// TIA Portal V17 export
// export: Created 2025-07-13T07:45:38.0095536Z, ExportSetting WithDefaults, DisplayName Totally Integrated Automation Portal, DisplayVersion V17, DisplayName TIA Portal Openness, DisplayVersion V17, DisplayName TIA Portal Version Control Interface, DisplayVersion V17, DisplayName STEP 7 Professional, DisplayVersion V17, DisplayName STEP 7 Safety, DisplayVersion V17, DisplayName WinCC Advanced / Unified PC, DisplayVersion V17
FUNCTION "valve_control" : Void   // FC4, LAD
{ S7_Optimized_Access := 'TRUE' }
VERSION : 0.1
// stored: AutoNumber true, IsIECCheckEnabled false, SetENOAutomatically false, UDAEnableTagReadback false
BEGIN

REGION Network 1
   // 1号电动阀
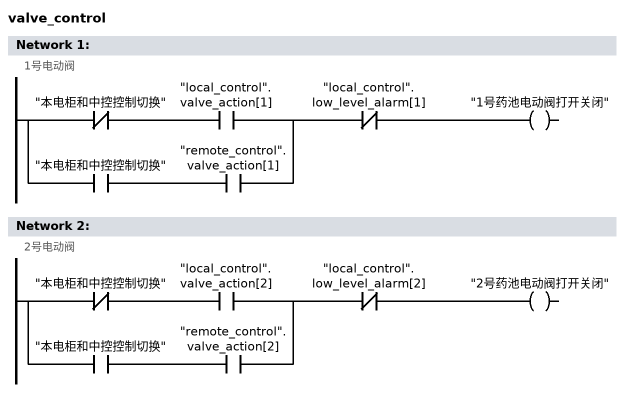
   RUNG wire#powerrail
      I_Contact( "本电柜和中控控制切换" )
      Contact( "local_control".valve_action[1] )
      wire#w1
      I_Contact( "local_control".low_level_alarm[1] )
      Coil( "1号药池电动阀打开关闭" )
   END_RUNG
   RUNG wire#powerrail
      Contact( "本电柜和中控控制切换" )
      Contact( "remote_control".valve_action[1] )
   END_RUNG wire#w1
   // the same network as SCL:
   "1号药池电动阀打开关闭" := ((NOT "本电柜和中控控制切换" AND "local_control".valve_action[1]) OR ("本电柜和中控控制切换" AND "remote_control".valve_action[1])) AND NOT "local_control".low_level_alarm[1];
END_REGION

REGION Network 2
   // 2号电动阀
   RUNG wire#powerrail
      I_Contact( "本电柜和中控控制切换" )
      Contact( "local_control".valve_action[2] )
      wire#w1
      I_Contact( "local_control".low_level_alarm[2] )
      Coil( "2号药池电动阀打开关闭" )
   END_RUNG
   RUNG wire#powerrail
      Contact( "本电柜和中控控制切换" )
      Contact( "remote_control".valve_action[2] )
   END_RUNG wire#w1
   // the same network as SCL:
   "2号药池电动阀打开关闭" := ((NOT "本电柜和中控控制切换" AND "local_control".valve_action[2]) OR ("本电柜和中控控制切换" AND "remote_control".valve_action[2])) AND NOT "local_control".low_level_alarm[2];
END_REGION
END_FUNCTION
